(* Logix 5000 project; controller L3 vendor 1 type 14 code 92 rev 20.12; software revision 20.04; part 9 of 9 *)
(* tags used below, declared in another part *)
   aux_dec : integrat;
   AUX_wkk5 : REAL;
   averagge_rate_sec : DINT;
   BITMW2 : BOOL;
   CV_PID_wkk : DINT;
   cv_pmpano : DINT;
   DateTime : DINT[7];   // DINT array tag for retrieve wallclock time through GSV created during conversion
   delta_cv_ano : DINT;
   delta_max_t_wkk : DINT;
   dif_I_red : DINT;
   diff_t_ano : DINT;
   fact_regul_pmpano : REAL;
   ForceStatus : INT;   // INT tag to retrieve Force enabled value through GSV created during conversion
   high_lim_pmpano : DINT;
   I_chut : BOOL;
   I_mont : BOOL;
   inc_ventilo : DINT;
   int_CV_wkk : integrat;
   L3_stat : DINT[20];
   L3_wkkk : DINT[125];
   low_lim_pmpano : DINT;
   mem1_i_tot : DINT;
   mem_cv_ano : DINT;
   mem_cv_pmpano : DINT;
   mem_i_tot : DINT;
   mem_t_ano : DINT;
   memtdec : REAL;
   N10 : DINT[233];
   N9 : DINT[200];   // niveau decapage vers lancy (n9[10) ;;N9[70]
   offstet_wkk : DINT;
   ons1 : BOOL;
   ons2 : BOOL;
   ons3 : BOOL;
   ons4 : BOOL;
   ons5 : BOOL;
   ons6 : BOOL;
   par_rate_en_sec : DINT;
   pid_dec_ch : PID;
   pid_dec_fr : PID;
   pid_pmpANO : PID;
   PIDwkk : PID;
   pmpano_inhold : BOOL;
   pmpano_inholdval : DINT;
   POS_V_COLO : DINT;
   POS_V_DEC : DINT;
   pour_offset_wkk : REAL;
   S : INT[164];
   S_C_TOUR : DINT;
   S_COND_TOUR : DINT;
   S_CSG_SPD_PMP_WKK : DINT;
   S_FLOW_TOUR : DINT;
   S_FLW_ech_DECAP : DINT;
   S_FLW_XCHG_DECAP : DINT;
   S_I_COL : DINT;
   S_I_COLO : DINT;
   S_I_R1 : DINT;
   S_I_R2 : DINT;
   S_I_R3 : DINT;
   S_I_R4 : DINT;
   S_IR1 : DINT;
   S_LVL_ANO : DINT;
   S_LVL_COLMAT : DINT;
   S_LVL_DECAP : DINT;
   S_LVL_NEUT : DINT;
   S_MA_PMP_WKK : BOOL;
   S_MAN_PMP_WKK : BOOL;
   S_niv_ANO : DINT;
   S_Q_PAS_NAOH : DINT;
   S_q_pass_h2so4 : DINT;
   S_SP_T_COLMAT : DINT;
   S_SPD_PMP_WKK : DINT;
   S_SPEED : DINT;
   S_T_ANO : DINT;
   S_T_AVER_COLM : DINT;
   S_T_COLO : DINT;
   S_T_DEC2 : DINT;
   S_T_DEC3 : REAL;
   S_T_DEGRAIS : DINT;
   S_T_EAU_REFROID : DINT;
   S_T_ent_COLM : DINT;
   S_T_IN_COLMAT : DINT;
   S_T_MID_COLMAT : DINT;
   S_T_moy_COLM : DINT;
   S_T_OUT_COLMAT : DINT;
   S_TEMPS_ANODIS : DINT;
   S_TEMPS_RUN_LINE : DINT;
   S_TEMPS_RUN_LINE_LAST_MONTH : DINT;
   S_TEMPS_STOP_LINE : DINT;
   S_TEMPS_STOP_LINE_LAST_MONTH : DINT;
   S_TOT_I : DINT;
   S_TPS_ANO_LAST_MONTH : DINT;
   S_TRACT : DINT;
   S_TRACT_BS3 : DINT;
   S_U_COLO : DINT;
   S_U_R1 : DINT;
   S_U_R2 : DINT;
   S_U_R3 : DINT;
   S_U_R4 : DINT;
   scp_CV_wkk : SCP;
   stat_L3 : DINT[20];
   Status : INT;   // INT tag to retrieve Status value through GSV created during conversion
   T4 : TIMER[180];
   t_seconde : TIMER;   // tempo on toutes les secondes
   vit_ventilo : DINT;
   wkk5 : REAL;
   wkk_L3 : DINT[125];
(* _2_GENERAL, continued *)

ROUTINE _9b_regul_ano   (* ladder *)
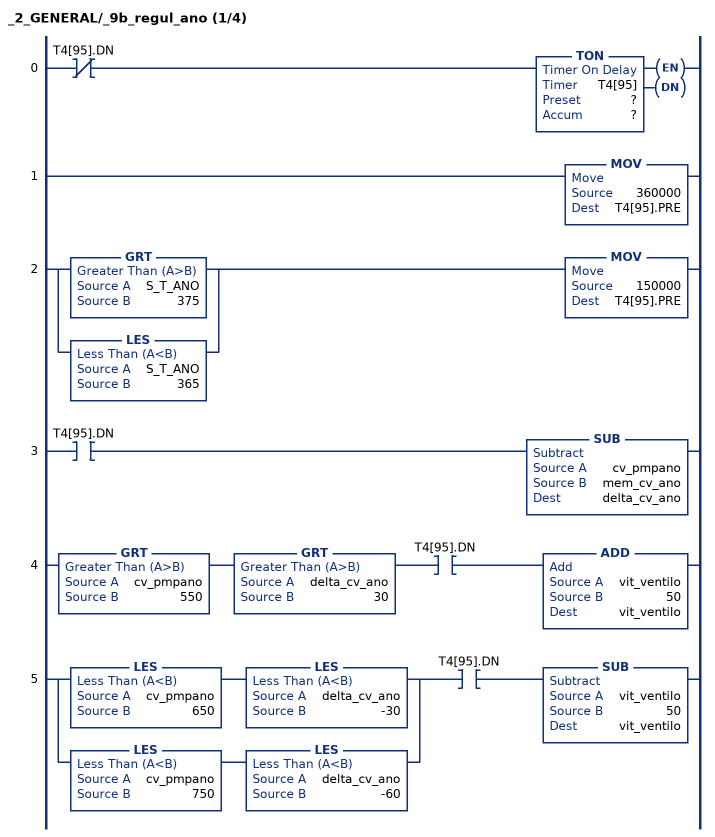
   0: XIO(T4[95].DN)TON(T4[95],?,?);
   1: MOV(360000,T4[95].PRE);
   2: [GRT(S_T_ANO,375) ,LES(S_T_ANO,365) ]MOV(150000,T4[95].PRE);
   3: XIC(T4[95].DN)SUB(cv_pmpano,mem_cv_ano,delta_cv_ano);
   4: GRT(cv_pmpano,550)GRT(delta_cv_ano,30)XIC(T4[95].DN)ADD(vit_ventilo,50,vit_ventilo);
   5: [LES(cv_pmpano,650) LES(delta_cv_ano,-30) ,LES(cv_pmpano,750) LES(delta_cv_ano,-60) ]XIC(T4[95].DN)SUB(vit_ventilo,50,vit_ventilo);
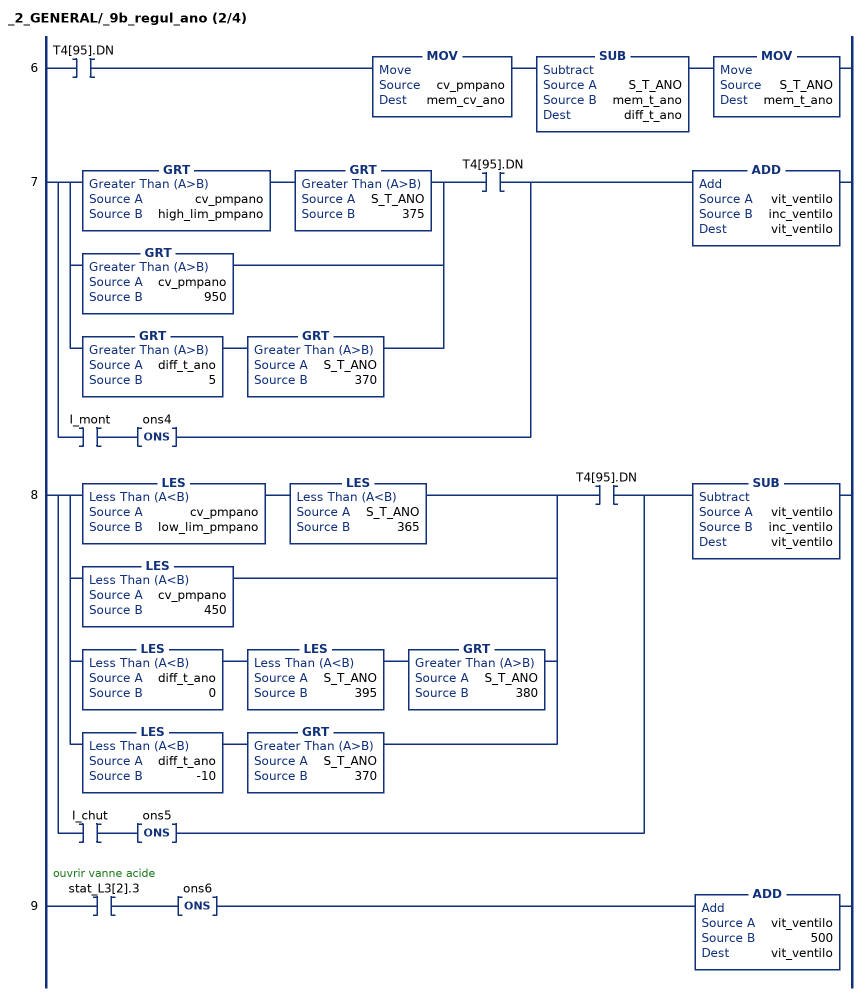
   6: XIC(T4[95].DN)MOV(cv_pmpano,mem_cv_ano)SUB(S_T_ANO,mem_t_ano,diff_t_ano)MOV(S_T_ANO,mem_t_ano);
   7: [[GRT(cv_pmpano,high_lim_pmpano) GRT(S_T_ANO,375) ,GRT(cv_pmpano,950) ,GRT(diff_t_ano,5) GRT(S_T_ANO,370) ] XIC(T4[95].DN) ,XIC(I_mont) ONS(ons4) ]ADD(vit_ventilo,inc_ventilo,vit_ventilo);
   8: [[LES(cv_pmpano,low_lim_pmpano) LES(S_T_ANO,365) ,LES(cv_pmpano,450) ,LES(diff_t_ano,0) LES(S_T_ANO,395) GRT(S_T_ANO,380) ,LES(diff_t_ano,-10) GRT(S_T_ANO,370) ] XIC(T4[95].DN) ,XIC(I_chut) ONS(ons5) ]SUB(vit_ventilo,inc_ventilo,vit_ventilo);
   9: XIC(stat_L3[2].3)ONS(ons6)ADD(vit_ventilo,500,vit_ventilo);
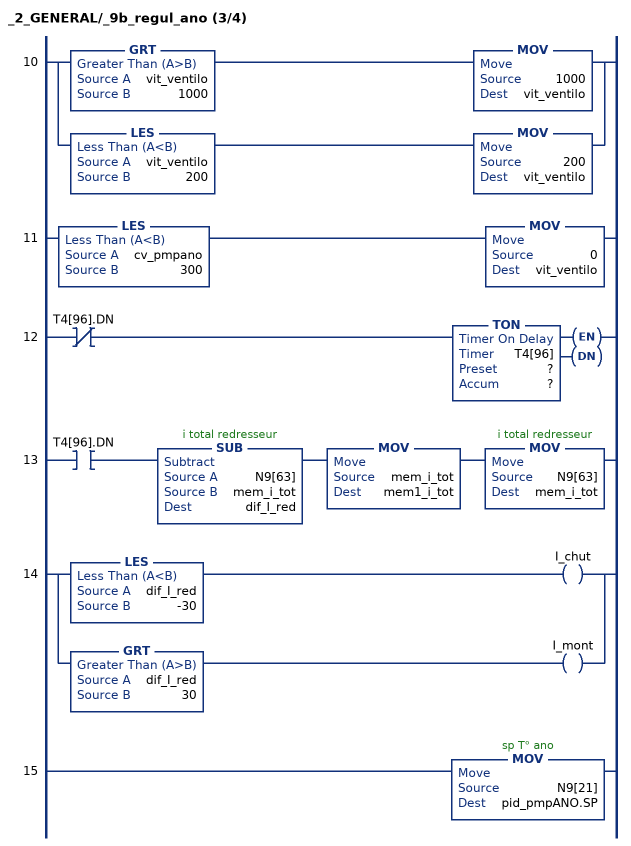
   10: [GRT(vit_ventilo,1000) MOV(1000,vit_ventilo) ,LES(vit_ventilo,200) MOV(200,vit_ventilo) ];
   11: LES(cv_pmpano,300)MOV(0,vit_ventilo);
   12: XIO(T4[96].DN)TON(T4[96],?,?);
   13: XIC(T4[96].DN)SUB(N9[63],mem_i_tot,dif_I_red)MOV(mem_i_tot,mem1_i_tot)MOV(N9[63],mem_i_tot);
   14: [LES(dif_I_red,-30) OTE(I_chut) ,GRT(dif_I_red,30) OTE(I_mont) ];
   15: MOV(N9[21],pid_pmpANO.SP);
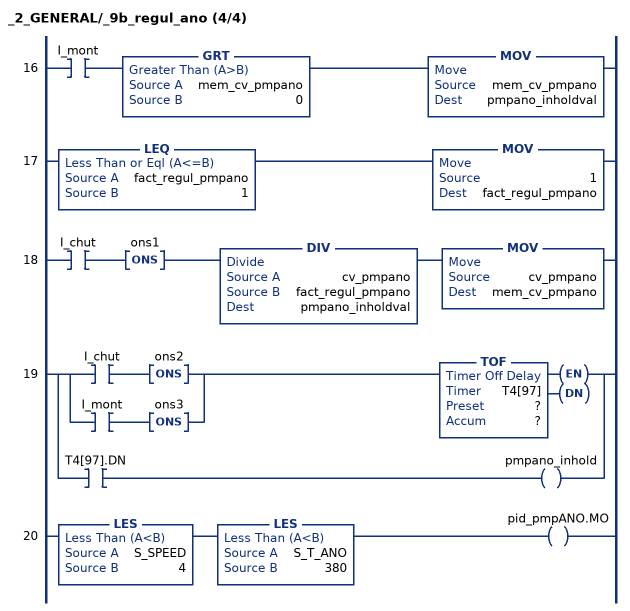
   16: XIC(I_mont)GRT(mem_cv_pmpano,0)MOV(mem_cv_pmpano,pmpano_inholdval);
   17: LEQ(fact_regul_pmpano,1)MOV(1,fact_regul_pmpano);
   18: XIC(I_chut)ONS(ons1)DIV(cv_pmpano,fact_regul_pmpano,pmpano_inholdval)MOV(cv_pmpano,mem_cv_pmpano);
   19: [[XIC(I_chut) ONS(ons2) ,XIC(I_mont) ONS(ons3) ] TOF(T4[97],?,?) ,XIC(T4[97].DN) OTE(pmpano_inhold) ];
   20: LES(S_SPEED,4)LES(S_T_ANO,380)OTE(pid_pmpANO.MO);
END_ROUTINE

ROUTINE apport_nitrique   (* ladder *)
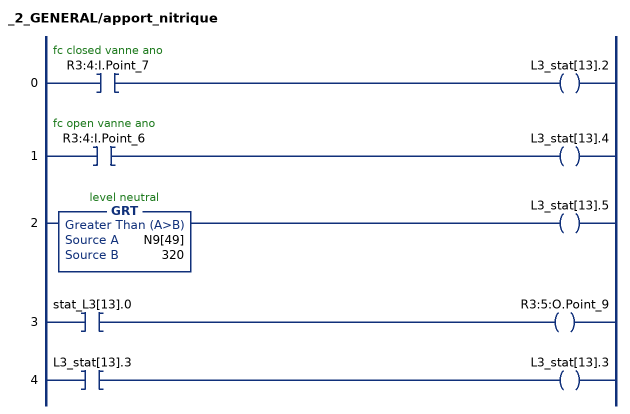
   0: XIC(R3:4:I.Point_7)OTE(L3_stat[13].2);
   1: XIC(R3:4:I.Point_6)OTE(L3_stat[13].4);
   2: GRT(N9[49],320)OTE(L3_stat[13].5);
   3: XIC(stat_L3[13].0)OTE(R3:5:O.Point_9);
   4: XIC(L3_stat[13].3)OTE(L3_stat[13].3);
END_ROUTINE

ROUTINE SUPERV   (* ladder *)
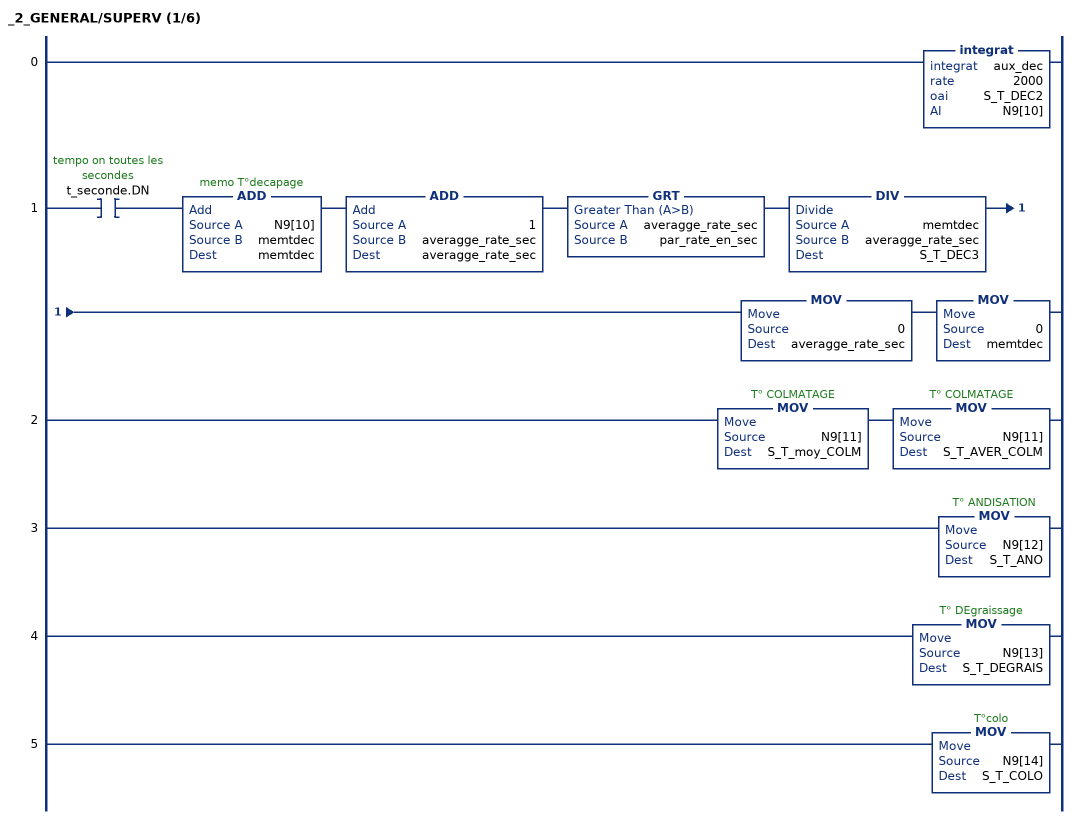
   0: integrat(aux_dec,2000,S_T_DEC2,N9[10]);
   1: XIC(t_seconde.DN)ADD(N9[10],memtdec,memtdec)ADD(1,averagge_rate_sec,averagge_rate_sec)GRT(averagge_rate_sec,par_rate_en_sec)DIV(memtdec,averagge_rate_sec,S_T_DEC3)MOV(0,averagge_rate_sec)MOV(0,memtdec);
   2: MOV(N9[11],S_T_moy_COLM)MOV(N9[11],S_T_AVER_COLM);
   3: MOV(N9[12],S_T_ANO);
   4: MOV(N9[13],S_T_DEGRAIS);
   5: MOV(N9[14],S_T_COLO);
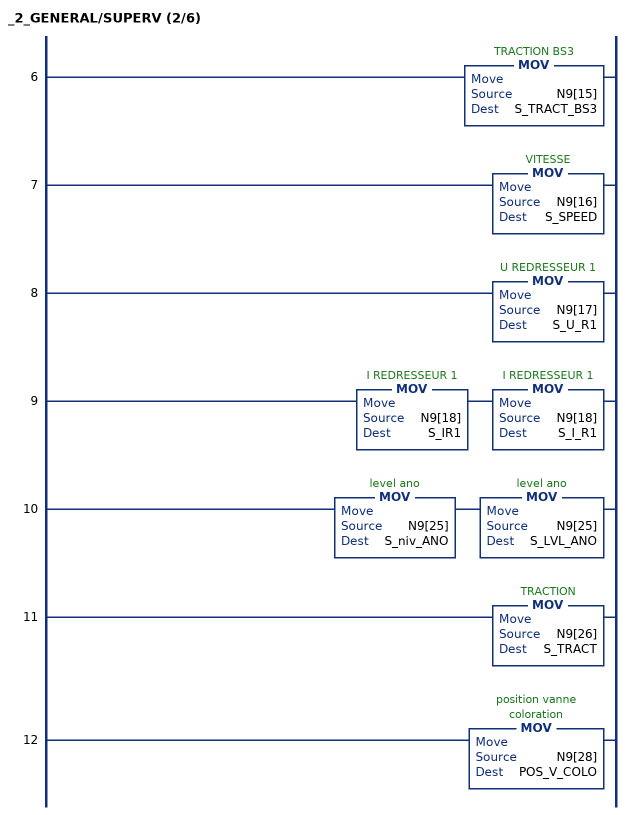
   6: MOV(N9[15],S_TRACT_BS3);
   7: MOV(N9[16],S_SPEED);
   8: MOV(N9[17],S_U_R1);
   9: MOV(N9[18],S_IR1)MOV(N9[18],S_I_R1);
   10: MOV(N9[25],S_niv_ANO)MOV(N9[25],S_LVL_ANO);
   11: MOV(N9[26],S_TRACT);
   12: MOV(N9[28],POS_V_COLO);
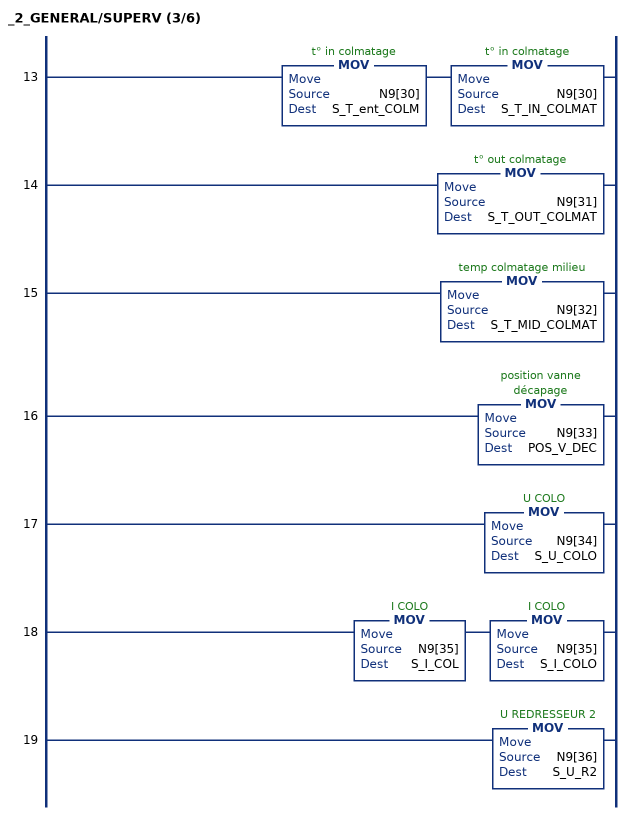
   13: MOV(N9[30],S_T_ent_COLM)MOV(N9[30],S_T_IN_COLMAT);
   14: MOV(N9[31],S_T_OUT_COLMAT);
   15: MOV(N9[32],S_T_MID_COLMAT);
   16: MOV(N9[33],POS_V_DEC);
   17: MOV(N9[34],S_U_COLO);
   18: MOV(N9[35],S_I_COL)MOV(N9[35],S_I_COLO);
   19: MOV(N9[36],S_U_R2);
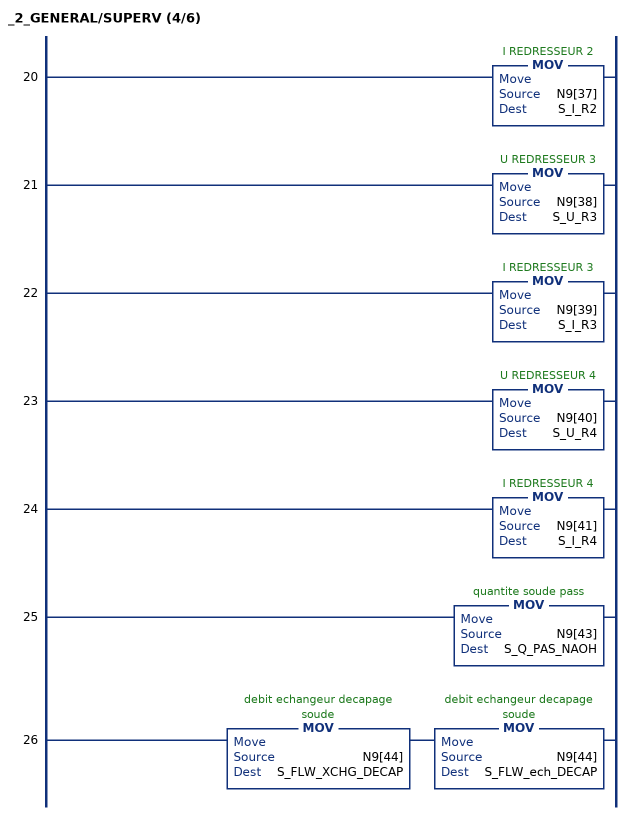
   20: MOV(N9[37],S_I_R2);
   21: MOV(N9[38],S_U_R3);
   22: MOV(N9[39],S_I_R3);
   23: MOV(N9[40],S_U_R4);
   24: MOV(N9[41],S_I_R4);
   25: MOV(N9[43],S_Q_PAS_NAOH);
   26: MOV(N9[44],S_FLW_XCHG_DECAP)MOV(N9[44],S_FLW_ech_DECAP);
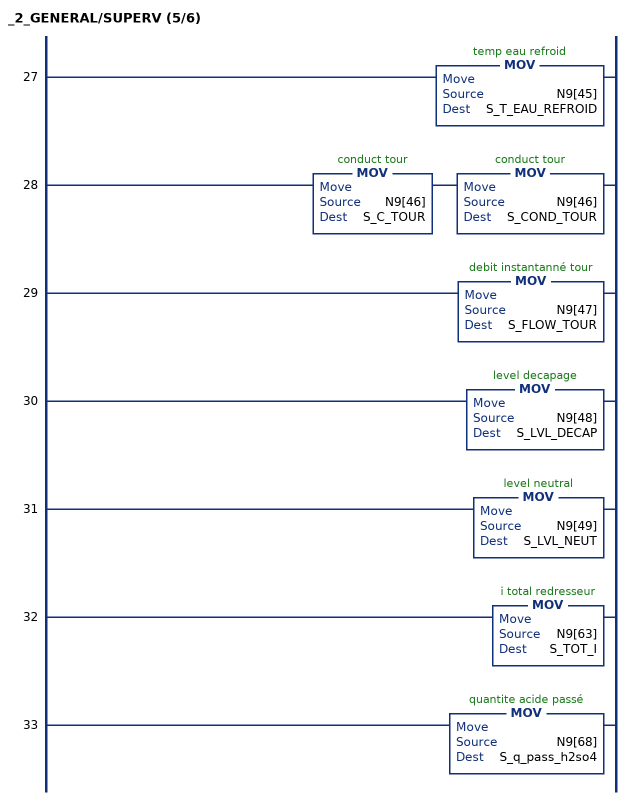
   27: MOV(N9[45],S_T_EAU_REFROID);
   28: MOV(N9[46],S_C_TOUR)MOV(N9[46],S_COND_TOUR);
   29: MOV(N9[47],S_FLOW_TOUR);
   30: MOV(N9[48],S_LVL_DECAP);
   31: MOV(N9[49],S_LVL_NEUT);
   32: MOV(N9[63],S_TOT_I);
   33: MOV(N9[68],S_q_pass_h2so4);
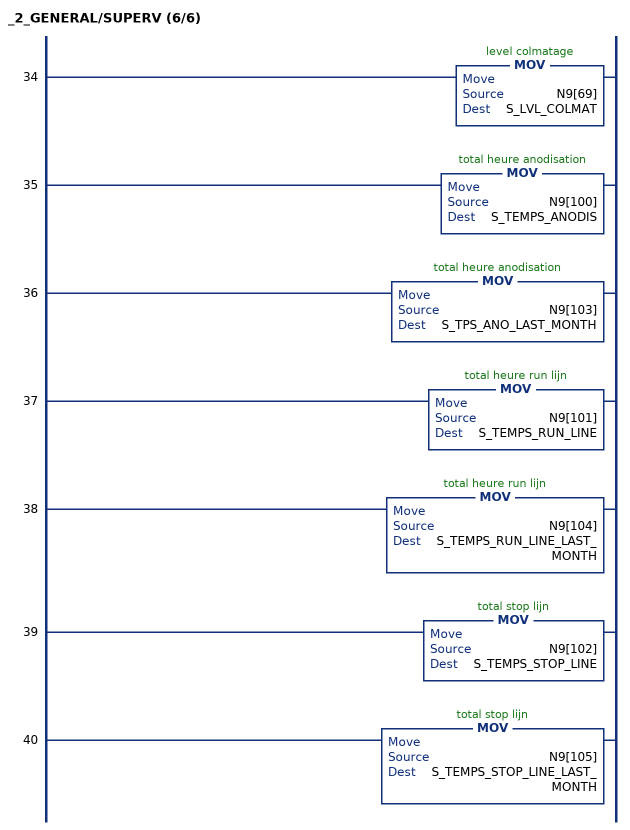
   34: MOV(N9[69],S_LVL_COLMAT);
   35: MOV(N9[100],S_TEMPS_ANODIS);
   36: MOV(N9[103],S_TPS_ANO_LAST_MONTH);
   37: MOV(N9[101],S_TEMPS_RUN_LINE);
   38: MOV(N9[104],S_TEMPS_RUN_LINE_LAST_MONTH);
   39: MOV(N9[102],S_TEMPS_STOP_LINE);
   40: MOV(N9[105],S_TEMPS_STOP_LINE_LAST_MONTH);
END_ROUTINE

ROUTINE wkk   (* ladder *)
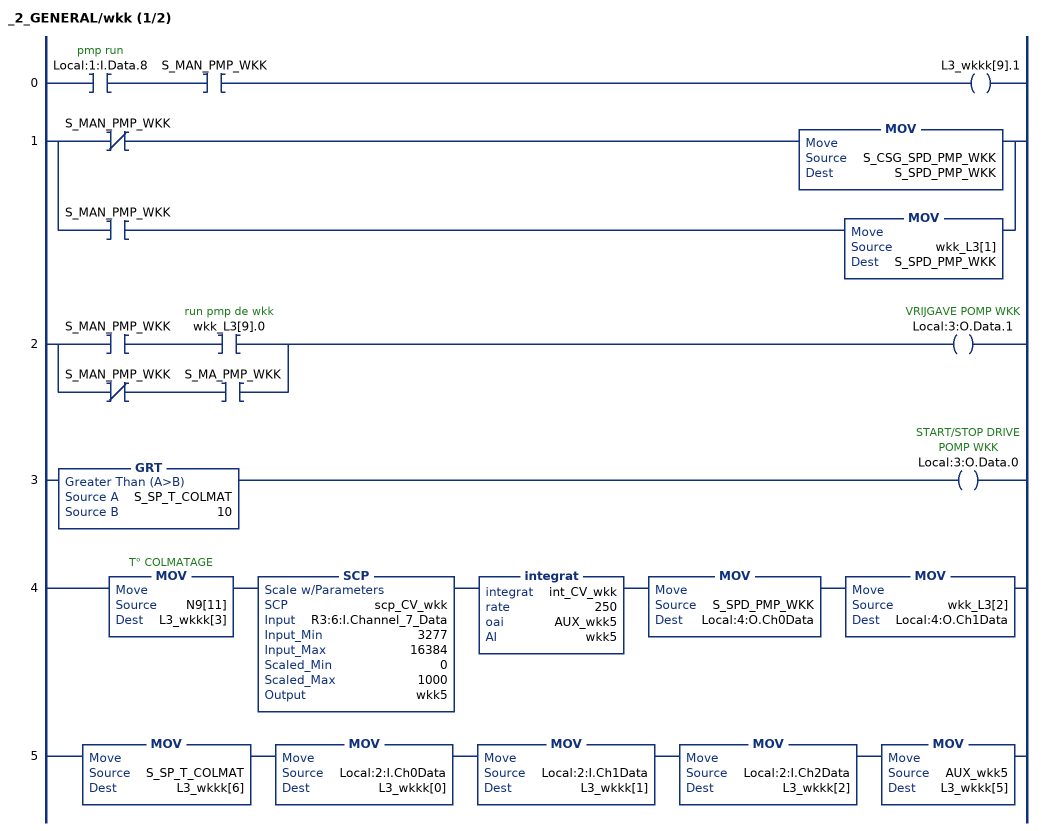
   0: XIC(Local:1:I.Data.8)XIC(S_MAN_PMP_WKK)OTE(L3_wkkk[9].1);
   1: [XIO(S_MAN_PMP_WKK) MOV(S_CSG_SPD_PMP_WKK,S_SPD_PMP_WKK) ,XIC(S_MAN_PMP_WKK) MOV(wkk_L3[1],S_SPD_PMP_WKK) ];
   2: [XIC(S_MAN_PMP_WKK) XIC(wkk_L3[9].0) ,XIO(S_MAN_PMP_WKK) XIC(S_MA_PMP_WKK) ]OTE(Local:3:O.Data.1);
   3: GRT(S_SP_T_COLMAT,10)OTE(Local:3:O.Data.0);
   4: MOV(N9[11],L3_wkkk[3])SCP(scp_CV_wkk,R3:6:I.Channel_7_Data,3277,16384,0,1000,wkk5)integrat(int_CV_wkk,250,AUX_wkk5,wkk5)MOV(S_SPD_PMP_WKK,Local:4:O.Ch0Data)MOV(wkk_L3[2],Local:4:O.Ch1Data);
   5: MOV(S_SP_T_COLMAT,L3_wkkk[6])MOV(Local:2:I.Ch0Data,L3_wkkk[0])MOV(Local:2:I.Ch1Data,L3_wkkk[1])MOV(Local:2:I.Ch2Data,L3_wkkk[2])MOV(AUX_wkk5,L3_wkkk[5]);
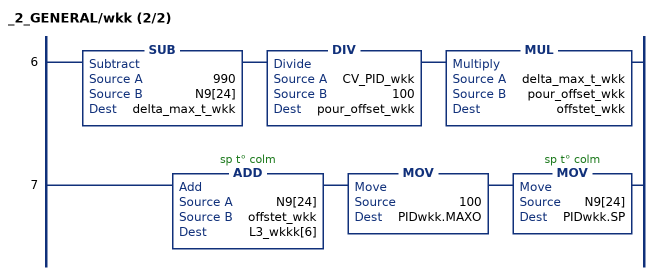
   6: SUB(990,N9[24],delta_max_t_wkk)DIV(CV_PID_wkk,100,pour_offset_wkk)MUL(delta_max_t_wkk,pour_offset_wkk,offstet_wkk);
   7: ADD(N9[24],offstet_wkk,L3_wkkk[6])MOV(100,PIDwkk.MAXO)MOV(N9[24],PIDwkk.SP);
END_ROUTINE
END_PROGRAM

PROGRAM MainProgram   (* main routine MainRoutine *)

ROUTINE MainRoutine   (* ladder *)
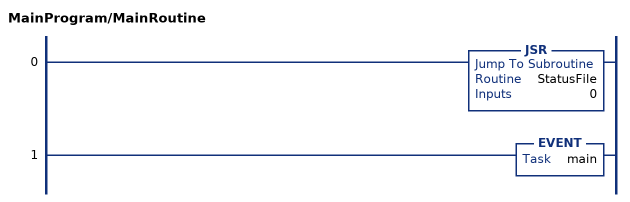
   0: JSR(StatusFile,0);
   1: EVENT(main);
END_ROUTINE

ROUTINE StatusFile   (* ladder *)
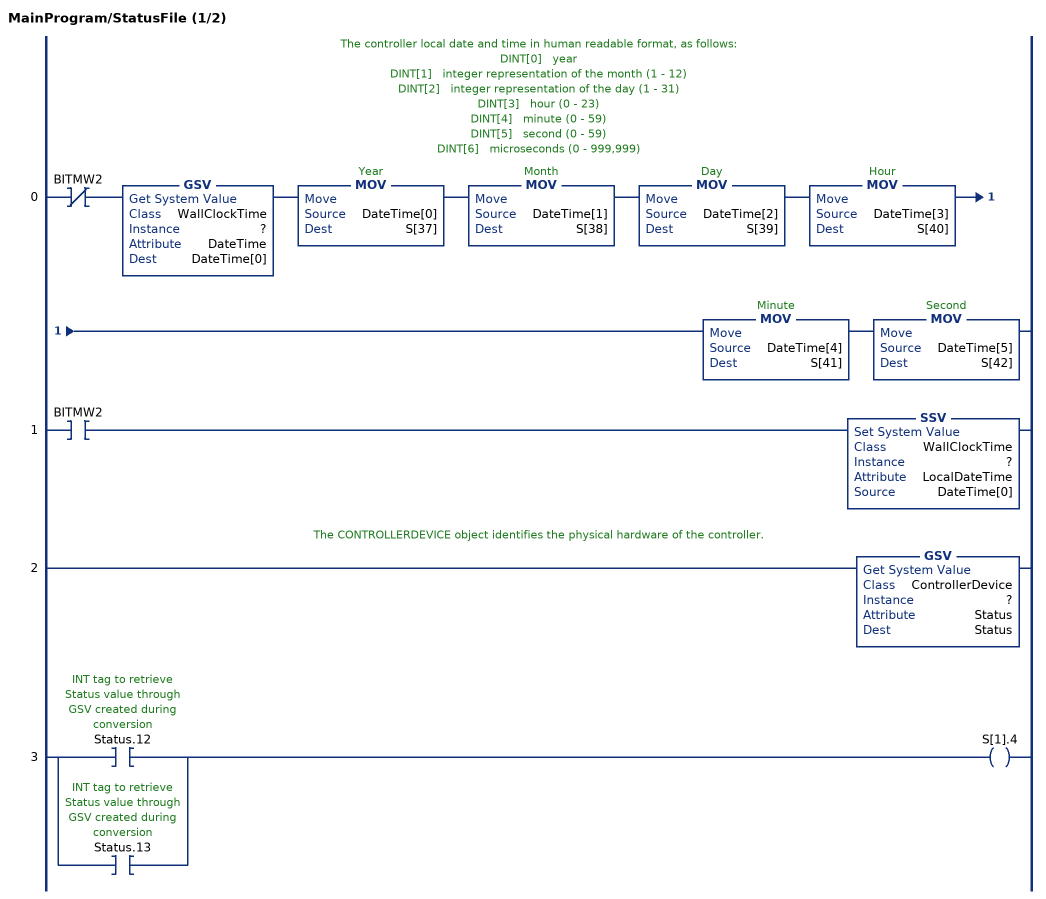
   // The controller local date and time in human readable format, as follows:
   // DINT[0] 	year
   // DINT[1] 	integer representation of the month (1 - 12)
   // DINT[2] 	integer representation of the day (1 - 31)
   // DINT[3] 	hour (0 - 23)
   // DINT[4] 	minute (0 - 59)
   // DINT[5] 	second (0 - 59)
   // DINT[6] 	microseconds (0 - 999,999)
   0: XIO(BITMW2)GSV(WallClockTime,?,DateTime,DateTime[0])MOV(DateTime[0],S[37])MOV(DateTime[1],S[38])MOV(DateTime[2],S[39])MOV(DateTime[3],S[40])MOV(DateTime[4],S[41])MOV(DateTime[5],S[42]);
   1: XIC(BITMW2)SSV(WallClockTime,?,LocalDateTime,DateTime[0]);
   // The CONTROLLERDEVICE object identifies the physical hardware of the controller.
   2: GSV(ControllerDevice,?,Status,Status);
   3: [XIC(Status.12) ,XIC(Status.13) ]OTE(S[1].4);
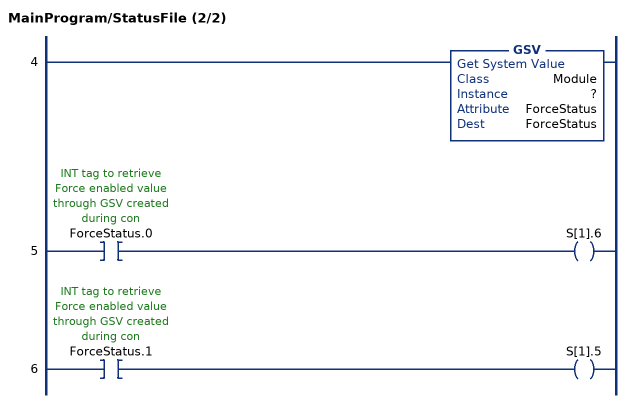
   4: GSV(Module,?,ForceStatus,ForceStatus);
   5: XIC(ForceStatus.0)OTE(S[1].6);
   6: XIC(ForceStatus.1)OTE(S[1].5);
END_ROUTINE
END_PROGRAM

PROGRAM pid_dec   (* main routine dec *)

ROUTINE dec   (* ladder *)
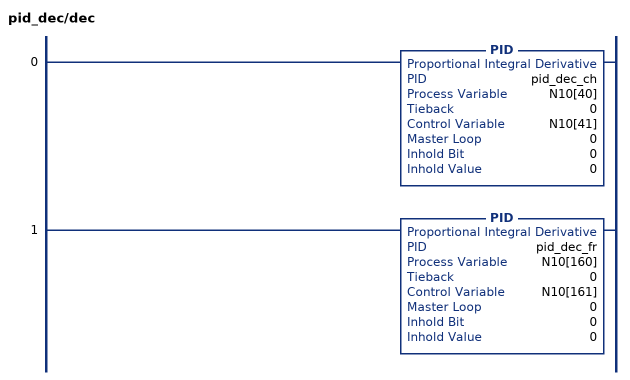
   0: PID(pid_dec_ch,N10[40],0,N10[41],0,0,0);
   1: PID(pid_dec_fr,N10[160],0,N10[161],0,0,0);
END_ROUTINE
END_PROGRAM
